{attribute 'qualified_only'}
VAR_GLOBAL
	B1: BOOL; // Schwimmerschalter oben
	B2: BOOL;     // Schwimmerschalter unten
	F1: BOOL;     // Thermorelais
	S1: BOOL;     // Wahlschalter Hand
	S2: BOOL;     // Wahlschalter Automatik
	S3: BOOL;      // Störung quittieren
END_VAR

(* stored: Version 1.1.0.1, ProductVersion 3.1.4024.5
   GVL SimDI: Id {c2d05302-d374-4f85-80dd-41006a3e3277} *)
